TYPE ST_AnalysisReset : 
STRUCT
	eResetComponent: E_AnalysisComponents := E_AnalysisComponents.All;
	bResetExecute: BOOL;
END_STRUCT
END_TYPE

(* stored: DUT ST_AnalysisReset: Id 390ee2e7-30db-4241-a98a-75f5546178da *)
